(*
SPDX-FileCopyrightText: © 2026 Oleksandr Tiutyk <trofimich@gmail.com>
SPDX-License-Identifier: MIT
License: https://opensource.org/license/mit
*)

{attribute 'qualified_only'}
{attribute 'strict'}
{attribute 'to_string'}
TYPE SORT_DIRECTION :
(
	ASCENDING,
	DESCENDING
);
END_TYPE

(* stored: Version 1.1.0.1
   DUT SORT_DIRECTION: Id {e7ff887b-998b-4e25-bad7-5430d7b7b13f} *)
